Staubli VAL3: listredraw.pgx

public program listRedraw(num x_nFirst)
begin
  //-----------------------------------------------------------------------
  //Header begin
  //Description of program
  //  Redraw the list in the userPage from the element number.
  //  pFirst of the list.
  //
  //Input parameters
  //  num x_nFirst :
  //    role : Defines the first element of the list
  //
  //Example
  //  call listRedraw(1)
  //
  //History
  //  Creation : 28-04-08 - f.Rob
  //Header end
  //-----------------------------------------------------------------------
  call listFrame(sTitle,nTopX,nTopY,nBottomX,nListHeight)
  call listUpdate(x_nFirst)
end
